FUNCTION_BLOCK TcoSequencerTestChildState EXTENDS TcoCore.TcoState
VAR
    _requestedState : UINT;
    _requestedStateCount : ULINT;
    _restoreCount : ULINT;
END_VAR

(*~
    <docu>
        <summary>
            This method is called on each change of the <c>State</c>. This method could be overloaded and custom code should be placed here.
        </summary>
    </docu>
~*)
METHOD PROTECTED OnStateChange
VAR_INPUT
    PreviousState : INT;
    NewState : INT;
END_VAR
IF NewState = _requestedState THEN
    _requestedStateCount := _requestedStateCount + 1;
END_IF

IF NewState = -1 THEN
    _restoreCount := _restoreCount + 1;
END_IF
END_METHOD

PROPERTY RequestedState : UINT
GET
RequestedState := _requestedState;
END_GET
SET
_requestedState := RequestedState;
END_SET
END_PROPERTY

END_FUNCTION_BLOCK

(* stored: Version 1.1.0.1
   POU TcoSequencerTestChildState: Id {47153bd6-c760-05f1-3cc8-dc997014292d}, SpecialFunc None
   Method OnStateChange: Id {405797a2-e34c-0ea1-11db-966029e7456c}
   Property RequestedState: Id {a41d472f-303d-05fb-1900-06b7f9599535}
   Get Get: Id {b556c158-7b7a-058d-2781-29d942d6c1f4}
   Set Set: Id {c6d0caec-be85-0b5b-3071-7596953df036} *)
